FUNCTION "fc_TEST_1" : Bool

{ S7_Optimized_Access := 'TRUE' }
VERSION : 0.1
VAR_INPUT

END_VAR

VAR_OUTPUT

END_VAR

VAR_IN_OUT

END_VAR

VAR_TEMP

END_VAR

VAR CONSTANT

END_VAR


BEGIN
	REGION INITIAL_FUNCTION
	    #fc_TEST_1 := TRUE;
	END_REGION

END_FUNCTION

